PROGRAM MAIN
VAR
	fb		: FB_MyBlock();
END_VAR

fb();

END_PROGRAM

(* stored: Version 1.1.0.1
   POU MAIN: Id {fa554e6f-e627-4186-9888-96357c6b05df}, SpecialFunc None *)
